KUKA KRL program: C3_mod.src

&ACCESS RVO
&PARAM EDITMASK = *
DEFFCT INT C3_mod(N:IN, M:IN)
   DECL INT N,M
   IF (N==0) OR (M==0) THEN
   RETURN 0
   ENDIF
   RETURN N-(N/M)*M
ENDFCT
